FUNCTION_BLOCK PUBLIC ramp
VAR_INPUT
	duration : INT;
	start_val : REAL;
	end_val : REAL;
	enable : BOOL;
END_VAR
VAR_OUTPUT
	output : REAL;
END_VAR
VAR
	ramp_tmr: TON;
	ramp_tmr_et: TIME;
	ramp_counter: CTU;
	ramp_time_delay_ms: real;
	ramp_time_delay: TIME;
	ramp_range : REAL;
	ramp_increment: REAL;
	ramp_tmr_et_ms: REAL;
	ramp_mult_output: REAL;
END_VAR

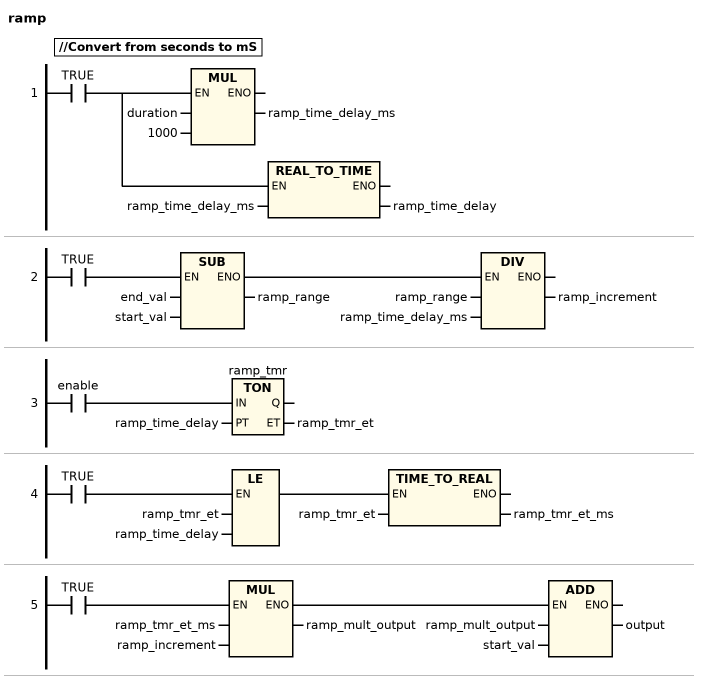
// NETWORK 1
// label: //Convert from seconds to mS
ramp_time_delay_ms := duration * 1000;
ramp_time_delay := REAL_TO_TIME(ramp_time_delay_ms);

// NETWORK 2
ramp_range := end_val - start_val;
ramp_increment := ramp_range / ramp_time_delay_ms;

// NETWORK 3
ramp_tmr(IN := enable, PT := ramp_time_delay, ET => ramp_tmr_et); // TON

// NETWORK 4
IF ramp_tmr_et <= ramp_time_delay THEN ramp_tmr_et_ms := TIME_TO_REAL(ramp_tmr_et); END_IF

// NETWORK 5
ramp_mult_output := ramp_tmr_et_ms * ramp_increment;
output := ramp_mult_output + start_val;

END_FUNCTION_BLOCK

(* stored: Version 1.1.0.1, ProductVersion 3.1.4024.12
   POU ramp: Id {e9094ae9-903d-4350-a822-9f015ddc92f3}, SpecialFunc None *)
